PROGRAM MAIN
VAR

	fb_Vereinzelung :FB_Vereinzelung;
	fb_EZylinder1 : FB_EZylinder;
	fb_EZylinder2 : FB_EZylinder;
	fb_Ampelleuchte :FB_Ampelleuchte;
	fb_Foerderband :FB_Foerderband;
	fb_Dispenser_Rot :FB_Dispenser;
	fb_Dispenser_Gruen :FB_Dispenser;
	fb_Dispenser_Blau :FB_Dispenser;
	
	
	
	value : Real;
	fb_Transport :FB_Transport;
END_VAR

value :=TO_UINT(FUN_Scale(4096,4096,0,350,0));



fb_Vereinzelung(
	bEnable:= IFC_HW.bEnable, 
	bExecute:= IFC_HW.bExecute, 
	bSens1:= IFC_HW.bEinzelSens1, 
	bSens2:= IFC_HW.bEinzelSens2, 
	bSens3:= IFC_HW.bEinzelSens3, 
	bSens4:= IFC_HW.bBandSens1, 
	eState=> , 
	bGate1=> fb_EZylinder1.bGate, 
	bGate2=> fb_EZylinder2.bGate);
	
fb_EZylinder1(bGate:= , bError:= , bR1=> IFC_HW.bR1AKT1, bR2=> IFC_HW.bR2AKT1);
fb_EZylinder2(bGate:= , bError:= , bR1=> IFC_HW.bR1AKT2, bR2=> IFC_HW.bR2AKT2);

//fb_Foerderband(
//	bEnable:= IFC_HW.bEnable, 
//	bExecute:= , 
//	bHalt:= , 
//	eState=> , 
//	ax:= IFC_HW.ax_BandMotor);
	
//fb_Dispenser_Rot(
//	bEnable:= IFC_HW.bEnable, 
//	bExecute:= , 
//	rDistance:= 60, 
//	eState=> , 
//	ax:= IFC_HW.ax_Extruder1);
	
//fb_Dispenser_Gruen(
//	bEnable:= IFC_HW.bEnable, 
//	bExecute:= IFC_HW.bBandSens2, 
//	rDistance:= 60, 
//	eState=> , 
//	ax:= IFC_HW.ax_Extruder2);
//	
//fb_Dispenser_Blau(
//	bEnable:= IFC_HW.bEnable, 
//	bExecute:= IFC_HW.bBandSens3, 
//	rDistance:= 60, 
//	eState=> , 
//	ax:= IFC_HW.ax_Extruder3);
//	


fb_Ampelleuchte(eState_Vereinzelung:= fb_Vereinzelung.eState, bAmpelGruen=> IFC_HW.bAmpelGrun, bAmpelRot=> IFC_HW.bAmpelRot, bAmpelGelb=> IFC_HW.bAmpelGelb);
	



//Transport als gesamtes
fb_Transport(
	bEnable:= IFC_HW.bEnable, 
	bExecute:= IFC_HW.bExecute, 
	nStation:= , 
	bSens1:= IFC_HW.bBandSens1, 
	bSens2:= IFC_HW.bBandSens2, 
	bSens3:= IFC_HW.bBandSens3, 
	bSens4:= IFC_HW.bBandSens4, 
	eState=> , 
	bStopper1=> IFC_HW.bBandHub1, 
	bStopper2=> IFC_HW.bBandHub2, 
	bStopper3=> IFC_HW.bBandHub3, 
	ax:= IFC_HW.ax_BandMotor);

END_PROGRAM

(* stored: Version 1.1.0.1, ProductVersion 3.1.4024.15
   POU MAIN: Id {bdcd83ff-4f15-4910-8ed3-f4b8d9a489d3}, SpecialFunc None *)
